// TIA Portal project "Pick_&_Place_XYZ_TIA_Portal" (V16)

(* hardware
DEVICE "S7-1200 station_1"  S7-1200 Station
   slot 0: "Rack_0"  S7-1200 Rack  Rack  V1.0
   slot 1: "PLC_1"  CPU 1215C DC/DC/DC  6ES7 215-1AG40-0XB0  V4.4
   slot 2: "DI 8x24VDC_1"  6ES7 221-1BF32-0XB0  V2.0
*)

// ===== PLC "PLC_1"  CPU 1215C DC/DC/DC =====

VAR_GLOBAL   // PLC tag table "Tabla de variables estándar"
   "pos_Y_alcanzada" AT %M0.6 : Bool;
   "pos_Z_alcanzada" AT %M0.7 : Bool;
   "Tag_1" AT %M500.3 : Bool;
   "Tag_2" AT %M200.0 : Bool;
   "arranque_cinta" AT %M1.0 : Bool;
END_VAR

VAR_GLOBAL   // PLC tag table "Entradas"
   "Box_at_place" AT %I2.0 : Bool;   // Sensor de posicion de lugar de carga del pale
   "Part_at_place" AT %I2.1 : Bool;   // Sensor de poscion de lugar de recogida de las cajas
   "Detected" AT %I2.2 : Bool;   // Sensor en la ventosa del robot cartesiano
   "C_limit" AT %I2.3 : Bool;   // Sensor que indica que la ventosa esta en angulo limite en giro en el eje Z
   "Start" AT %I2.4 : Bool;   // Pulsador de start
   "Reset" AT %I2.5 : Bool;   // Pulsador de reset
   "Stop" AT %I2.6 : Bool;   // Pulsador de stop
   "Emergency_stop" AT %I2.7 : Bool;   // Seta de emergencia
   "Auto" AT %I3.0 : Bool;   // Selector rotativo en posicion auto
   "X" AT %ID100 : Real;   // Coordenada X del robot, realimentada
   "Y" AT %ID104 : Real;   // Coordenada Y del robot, realimentada
   "Z" AT %ID108 : Real;   // Coordenada Z del robot, realimentada
END_VAR

VAR_GLOBAL   // PLC tag table "Salidas"
   "Box_conveyor" AT %Q0.0 : Bool;   // Cinta de rodillo para los pales
   "Part_conveyor" AT %Q0.1 : Bool;   // Cinta para las cajas
   "Exit_conveyor" AT %Q0.2 : Bool;   // Cinta de rodillo para salida de pales con cajas
   "C+" AT %Q0.3 : Bool;   // Actuador de giro de la ventosa, sentido horario mirando desde arriba
   "Grab" AT %Q0.4 : Bool;   // Ventosa
   "Exit_green" AT %Q0.5 : Bool;   // Semaforo industrial, color verde
   "Exit_yellow" AT %Q0.6 : Bool;   // Semaforo industrial, color amarillo
   "Exit_red" AT %Q0.7 : Bool;   // Semaforo industrial, color rojo
   "Start_light" AT %Q1.0 : Bool;   // Luz de pulsador de start
   "Reset_light" AT %Q1.1 : Bool;   // Luz de pulsador de reset
   "Stop_light" AT %Q1.2 : Bool;   // Luz de pulsador de stop
   "SP_X" AT %QD100 : Real;   // Salida de posicion del eje X del robot cartesiano
   "SP_Y" AT %QD104 : Real;   // Salida de posicion del eje Y del robot cartesiano
   "SP_Z" AT %QD108 : Real;   // Salida de posicion del eje Z del robor cartesiano
   "Counter" AT %QD112 : DInt;   // Display numerico para contador
END_VAR

VAR_GLOBAL   // PLC tag table "variables_auxiliares"
   "FlancoP_sensor_pales" AT %M10.0 : Bool;
   "Marcha" AT %M0.0 : Bool;
   "FlancoN_sensor_pales" AT %M500.0 : Bool;
   "Set_box_conveyor" AT %M500.1 : Bool;
   "FlancoP_estado_marcha" AT %M500.2 : Bool;
   "pale_terminado" AT %M0.1 : Bool;
   "Stop_filtrado" AT %M0.2 : Bool;
   "pos_X_alcanzada" AT %M0.5 : Bool;
   "caja_preparada" AT %M0.3 : Bool;
   "pale_preparado" AT %M0.4 : Bool;
END_VAR

TYPE "posicion_robot"
   STRUCT
      X : Real;
      Y : Real;
      Z : Real;
   END_STRUCT;
END_TYPE

// folder: DBs

DATA_BLOCK "contador_terminados_DB"   // DB1
{ S7_Optimized_Access := 'TRUE' }
VERSION : 0.1
// stored: InstanceOfName contador_terminados
"contador_terminados"
BEGIN
END_DATA_BLOCK

DATA_BLOCK "control_robot_y_ciclo_DB"   // DB2
{ S7_Optimized_Access := 'TRUE' }
VERSION : 0.1
// stored: InstanceOfName control_robot_y_ciclo
"control_robot_y_ciclo"
BEGIN
END_DATA_BLOCK

DATA_BLOCK "posiciones_robot"   // DB3
{ S7_Optimized_Access := 'TRUE' }
VERSION : 0.1
   VAR
      home : "posicion_robot";
      coger_caja_aprox : "posicion_robot";
      coger_caja : "posicion_robot";
      dejar_caja_1_aprox : "posicion_robot";
      dejar_caja_1 : "posicion_robot";
      dejar_caja_2_aprox : "posicion_robot";
      dejar_caja_2 : "posicion_robot";
      dejar_caja_3_aprox : "posicion_robot";
      dejar_caja_3 : "posicion_robot";
   END_VAR
BEGIN
   home.Y := 0.0;
   home.X := 0.0;
   home.Z := 0.0;
   coger_caja.X := 7.7;
   coger_caja.Y := 5.6;
   coger_caja.Z := 5.0;
   coger_caja_aprox.X := 7.7;
   coger_caja_aprox.Y := 5.6;
   coger_caja_aprox.Z := 0.0;
   dejar_caja_1_aprox.Y := 5.0;
   dejar_caja_1_aprox.Z := 0.0;
   dejar_caja_1.Z := 10.0;
   dejar_caja_1.Y := 5.0;
   dejar_caja_1_aprox.X := 2.5;
   dejar_caja_1.X := 2.5;
   dejar_caja_2.X := 4.2;
   dejar_caja_2.Y := 5.0;
   dejar_caja_2.Z := 10.0;
   dejar_caja_2_aprox.Z := 0.0;
   dejar_caja_2_aprox.Y := 5.0;
   dejar_caja_2_aprox.X := 4.2;
   dejar_caja_3.Y := 5.0;
   dejar_caja_3_aprox.Y := 5.0;
   dejar_caja_3_aprox.Z := 0.0;
   dejar_caja_3_aprox.X := 3.3;
   dejar_caja_3.X := 3.3;
   dejar_caja_3.Z := 5.5;
END_DATA_BLOCK

// folder: Conexion_factoryIO

FUNCTION "MHJ-PLC-Lab-Function-S71200" : Void   // FC9000, SCL
{ S7_Optimized_Access := 'TRUE' }
VERSION : 0.1
   VAR_TEMP
      rdTimeReturn : Int;
      outputTime : DTL;
      SyncVal : Byte;
      forVal : Int;
      forVal_2 : Int;
      Value : Byte;
   END_VAR
   VAR CONSTANT
      CompVal : Byte := 16#34;
      Value_01 : Byte := 16#11;
      Value_01_DW : DWord := 16#A165_D992;
      Value_02_DW : DWord := 16#58BE_4401;
   END_VAR
BEGIN

   #Value:=PEEK(area := 16#82,
        dbNumber := 0,
        byteOffset := 511);
   #Value := #Value + 1;

   POKE(area := 16#82,
        dbNumber := 0,
        byteOffset := 511,
        value := #Value);

   POKE(area:=16#81,
        dbNumber:=0,
        byteOffset:=1016,
        value:=#Value_01_DW);
   POKE(area := 16#81,
        dbNumber := 0,
        byteOffset := 1020,
        value := #Value_02_DW);

   POKE(area := 16#81,
        dbNumber := 0,
        byteOffset := 511,
        value := B#16#00);

   FOR #forVal := 0 TO 120 DO
       FOR #forVal_2:=0 TO 10 DO
           #rdTimeReturn:=RD_SYS_T(#outputTime);
           #rdTimeReturn := WR_SYS_T(#outputTime);
           #rdTimeReturn := RD_SYS_T(#outputTime);
           #rdTimeReturn := WR_SYS_T(#outputTime);
       END_FOR;
       #SyncVal:= PEEK(area := 16#81,
                      dbNumber := 0,
                      byteOffset := 511);
       IF #SyncVal = #CompVal THEN
          GOTO M_1;
       END_IF;
   END_FOR;
   RETURN;

   M_1:
   POKE(area := 16#81,
        dbNumber := 0,
        byteOffset := 511,
        value := B#16#0);
END_FUNCTION

// folder: FBs

FUNCTION_BLOCK "contador_terminados"   // FB1, LAD
{ S7_Optimized_Access := 'TRUE' }
VERSION : 0.1
   VAR RETAIN
      Contador_terminados : CTU_INT;
   END_VAR
   VAR_TEMP   // added for the SCL form of the ladder/FBD networks
      _w1 : Bool;
   END_VAR
BEGIN

REGION Network 1: Contador que incrementa con el flanco positivo de sesnsor NC, osea cuando el pale se va
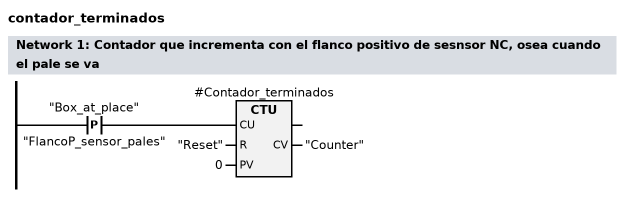
   #_w1 := "Box_at_place" AND NOT "FlancoP_sensor_pales";   // rising edge of "Box_at_place"
   "FlancoP_sensor_pales" := "Box_at_place";
   #Contador_terminados(CU := #_w1, R := "Reset", PV := 0, CV => "Counter");   // CTU
END_REGION
END_FUNCTION_BLOCK

FUNCTION_BLOCK "control_robot_y_ciclo"   // FB2, LAD
{ S7_Optimized_Access := 'TRUE' }
VERSION : 0.1
   VAR
      E0 : Bool;
      E1 : Bool;
      E2 : Bool;
      E3 : Bool;
      E4 : Bool;
      E5 : Bool;
      E6 : Bool;
      E7 : Bool;
      E8 : Bool;
      E9 : Bool;
      E10 : Bool;
      E11 : Bool;
      E12 : Bool;
      E13 : Bool;
      E14 : Bool;
      E15 : Bool;
      E16 : Bool;
      E17 : Bool;
      E18 : Bool;
      E19 : Bool;
      E20 : Bool;
      E21 : Bool;
      E22 : Bool;
      pos_X_alcanzada : Bool;
      pos_Y_alcanzada : Bool;
      pos_Z_alcanzada : Bool;
      aux1 : Bool;
      aux2 : Bool;
      aux3 : Bool;
      aux4 : Bool;
      aux5 : Bool;
      TON_1 : TON_TIME;
      TON_2 : TON_TIME;
      TON_3 : TON_TIME;
      TON_4 : TON_TIME;
   END_VAR
   VAR_TEMP   // added for the SCL form of the ladder/FBD networks
      _w1 : Bool;
      _w2 : Bool;
      _w3 : Bool;
      _w4 : Bool;
      _w5 : Bool;
      _w6 : Bool;
      _w7 : Bool;
   END_VAR
BEGIN

REGION Network 1
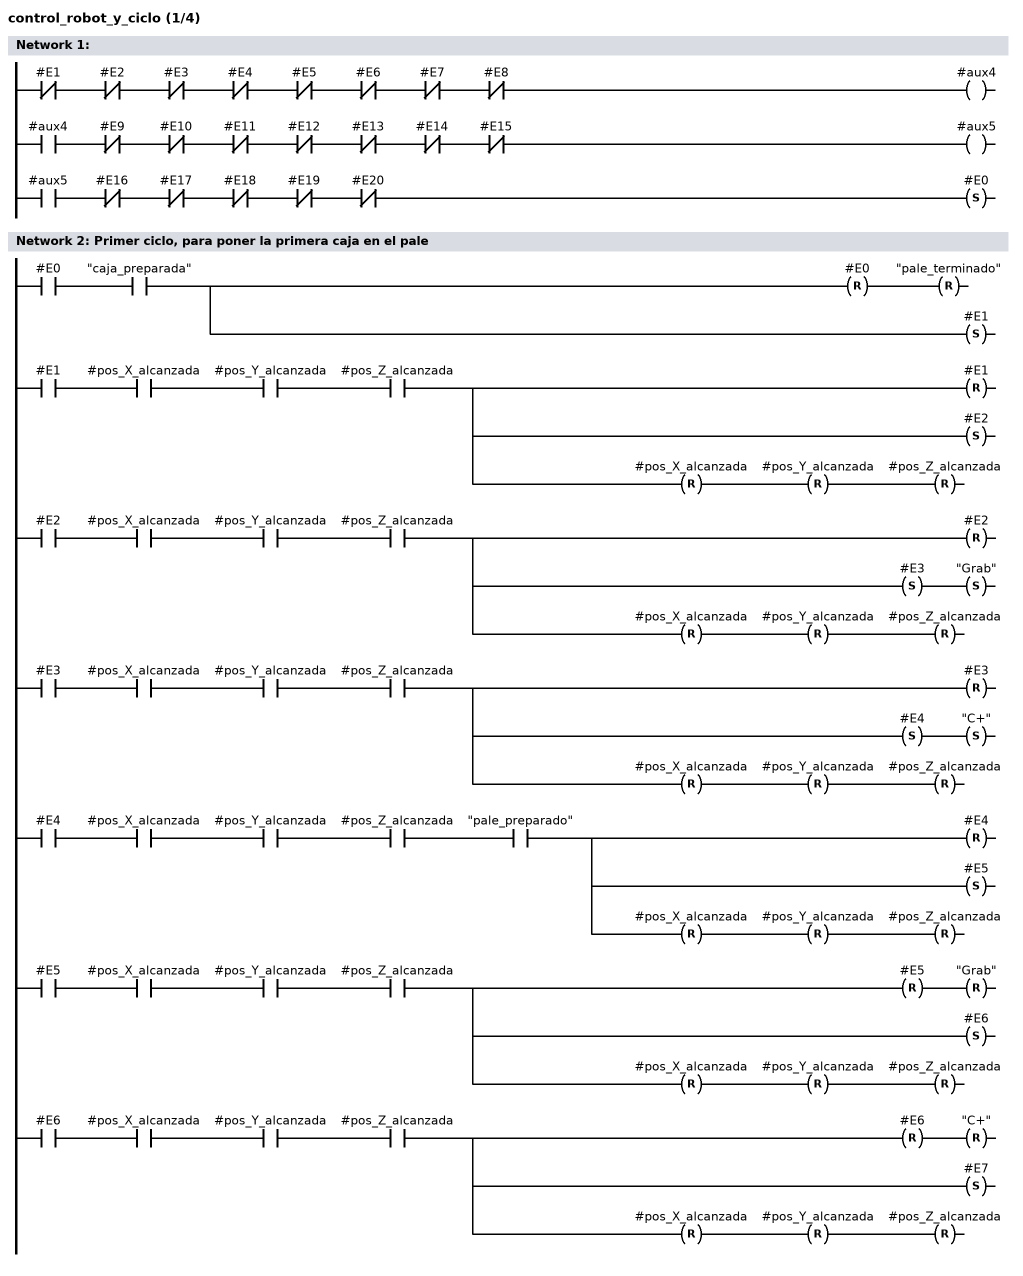
   RUNG wire#powerrail
      I_Contact( #E1 )
      I_Contact( #E2 )
      I_Contact( #E3 )
      I_Contact( #E4 )
      I_Contact( #E5 )
      I_Contact( #E6 )
      I_Contact( #E7 )
      I_Contact( #E8 )
      Coil( #aux4 )
   END_RUNG
   RUNG wire#powerrail
      Contact( #aux4 )
      I_Contact( #E9 )
      I_Contact( #E10 )
      I_Contact( #E11 )
      I_Contact( #E12 )
      I_Contact( #E13 )
      I_Contact( #E14 )
      I_Contact( #E15 )
      Coil( #aux5 )
   END_RUNG
   RUNG wire#powerrail
      Contact( #aux5 )
      I_Contact( #E16 )
      I_Contact( #E17 )
      I_Contact( #E18 )
      I_Contact( #E19 )
      I_Contact( #E20 )
      S_Coil( #E0 )
   END_RUNG
   // the same network as SCL:
   #aux4 := NOT #E1 AND NOT #E2 AND NOT #E3 AND NOT #E4 AND NOT #E5 AND NOT #E6 AND NOT #E7 AND NOT #E8;
   #aux5 := #aux4 AND NOT #E9 AND NOT #E10 AND NOT #E11 AND NOT #E12 AND NOT #E13 AND NOT #E14 AND NOT #E15;
   IF #aux5 AND NOT #E16 AND NOT #E17 AND NOT #E18 AND NOT #E19 AND NOT #E20 THEN #E0 := TRUE; END_IF;
END_REGION

REGION Network 2: Primer ciclo, para poner la primera caja en el pale
   RUNG wire#powerrail
      Contact( #E0 )
      Contact( "caja_preparada" )
      wire#w1
      R_Coil( #E0 )
      R_Coil( "pale_terminado" )
   END_RUNG
   RUNG wire#w1
      S_Coil( #E1 )
   END_RUNG
   RUNG wire#powerrail
      Contact( #E1 )
      Contact( #pos_X_alcanzada )
      Contact( #pos_Y_alcanzada )
      Contact( #pos_Z_alcanzada )
      wire#w2
      R_Coil( #E1 )
   END_RUNG
   RUNG wire#w2
      S_Coil( #E2 )
   END_RUNG
   RUNG wire#w2
      R_Coil( #pos_X_alcanzada )
      R_Coil( #pos_Y_alcanzada )
      R_Coil( #pos_Z_alcanzada )
   END_RUNG
   RUNG wire#powerrail
      Contact( #E2 )
      Contact( #pos_X_alcanzada )
      Contact( #pos_Y_alcanzada )
      Contact( #pos_Z_alcanzada )
      wire#w3
      R_Coil( #E2 )
   END_RUNG
   RUNG wire#w3
      S_Coil( #E3 )
      S_Coil( "Grab" )
   END_RUNG
   RUNG wire#w3
      R_Coil( #pos_X_alcanzada )
      R_Coil( #pos_Y_alcanzada )
      R_Coil( #pos_Z_alcanzada )
   END_RUNG
   RUNG wire#powerrail
      Contact( #E3 )
      Contact( #pos_X_alcanzada )
      Contact( #pos_Y_alcanzada )
      Contact( #pos_Z_alcanzada )
      wire#w4
      R_Coil( #E3 )
   END_RUNG
   RUNG wire#w4
      S_Coil( #E4 )
      S_Coil( "C+" )
   END_RUNG
   RUNG wire#w4
      R_Coil( #pos_X_alcanzada )
      R_Coil( #pos_Y_alcanzada )
      R_Coil( #pos_Z_alcanzada )
   END_RUNG
   RUNG wire#powerrail
      Contact( #E4 )
      Contact( #pos_X_alcanzada )
      Contact( #pos_Y_alcanzada )
      Contact( #pos_Z_alcanzada )
      Contact( "pale_preparado" )
      wire#w5
      R_Coil( #E4 )
   END_RUNG
   RUNG wire#w5
      S_Coil( #E5 )
   END_RUNG
   RUNG wire#w5
      R_Coil( #pos_X_alcanzada )
      R_Coil( #pos_Y_alcanzada )
      R_Coil( #pos_Z_alcanzada )
   END_RUNG
   RUNG wire#powerrail
      Contact( #E5 )
      Contact( #pos_X_alcanzada )
      Contact( #pos_Y_alcanzada )
      Contact( #pos_Z_alcanzada )
      wire#w6
      R_Coil( #E5 )
      R_Coil( "Grab" )
   END_RUNG
   RUNG wire#w6
      S_Coil( #E6 )
   END_RUNG
   RUNG wire#w6
      R_Coil( #pos_X_alcanzada )
      R_Coil( #pos_Y_alcanzada )
      R_Coil( #pos_Z_alcanzada )
   END_RUNG
   RUNG wire#powerrail
      Contact( #E6 )
      Contact( #pos_X_alcanzada )
      Contact( #pos_Y_alcanzada )
      Contact( #pos_Z_alcanzada )
      wire#w7
      R_Coil( #E6 )
      R_Coil( "C+" )
   END_RUNG
   RUNG wire#w7
      S_Coil( #E7 )
   END_RUNG
   RUNG wire#w7
      R_Coil( #pos_X_alcanzada )
      R_Coil( #pos_Y_alcanzada )
      R_Coil( #pos_Z_alcanzada )
   END_RUNG
   // the same network as SCL:
   #_w1 := #E0 AND "caja_preparada";
   IF #_w1 THEN
       #E0 := FALSE;
       "pale_terminado" := FALSE;
       #E1 := TRUE;
   END_IF;
   #_w2 := #E1 AND #pos_X_alcanzada AND #pos_Y_alcanzada AND #pos_Z_alcanzada;
   IF #_w2 THEN
       #E1 := FALSE;
       #E2 := TRUE;
       #pos_X_alcanzada := FALSE;
       #pos_Y_alcanzada := FALSE;
       #pos_Z_alcanzada := FALSE;
   END_IF;
   #_w3 := #E2 AND #pos_X_alcanzada AND #pos_Y_alcanzada AND #pos_Z_alcanzada;
   IF #_w3 THEN
       #E2 := FALSE;
       #E3 := TRUE;
       "Grab" := TRUE;
       #pos_X_alcanzada := FALSE;
       #pos_Y_alcanzada := FALSE;
       #pos_Z_alcanzada := FALSE;
   END_IF;
   #_w4 := #E3 AND #pos_X_alcanzada AND #pos_Y_alcanzada AND #pos_Z_alcanzada;
   IF #_w4 THEN
       #E3 := FALSE;
       #E4 := TRUE;
       "C+" := TRUE;
       #pos_X_alcanzada := FALSE;
       #pos_Y_alcanzada := FALSE;
       #pos_Z_alcanzada := FALSE;
   END_IF;
   #_w5 := #E4 AND #pos_X_alcanzada AND #pos_Y_alcanzada AND #pos_Z_alcanzada AND "pale_preparado";
   IF #_w5 THEN
       #E4 := FALSE;
       #E5 := TRUE;
       #pos_X_alcanzada := FALSE;
       #pos_Y_alcanzada := FALSE;
       #pos_Z_alcanzada := FALSE;
   END_IF;
   #_w6 := #E5 AND #pos_X_alcanzada AND #pos_Y_alcanzada AND #pos_Z_alcanzada;
   IF #_w6 THEN
       #E5 := FALSE;
       "Grab" := FALSE;
       #E6 := TRUE;
       #pos_X_alcanzada := FALSE;
       #pos_Y_alcanzada := FALSE;
       #pos_Z_alcanzada := FALSE;
   END_IF;
   #_w7 := #E6 AND #pos_X_alcanzada AND #pos_Y_alcanzada AND #pos_Z_alcanzada;
   IF #_w7 THEN
       #E6 := FALSE;
       "C+" := FALSE;
       #E7 := TRUE;
       #pos_X_alcanzada := FALSE;
       #pos_Y_alcanzada := FALSE;
       #pos_Z_alcanzada := FALSE;
   END_IF;
END_REGION

REGION Network 3: segundo ciclo, para poner la segunda caja en el pale
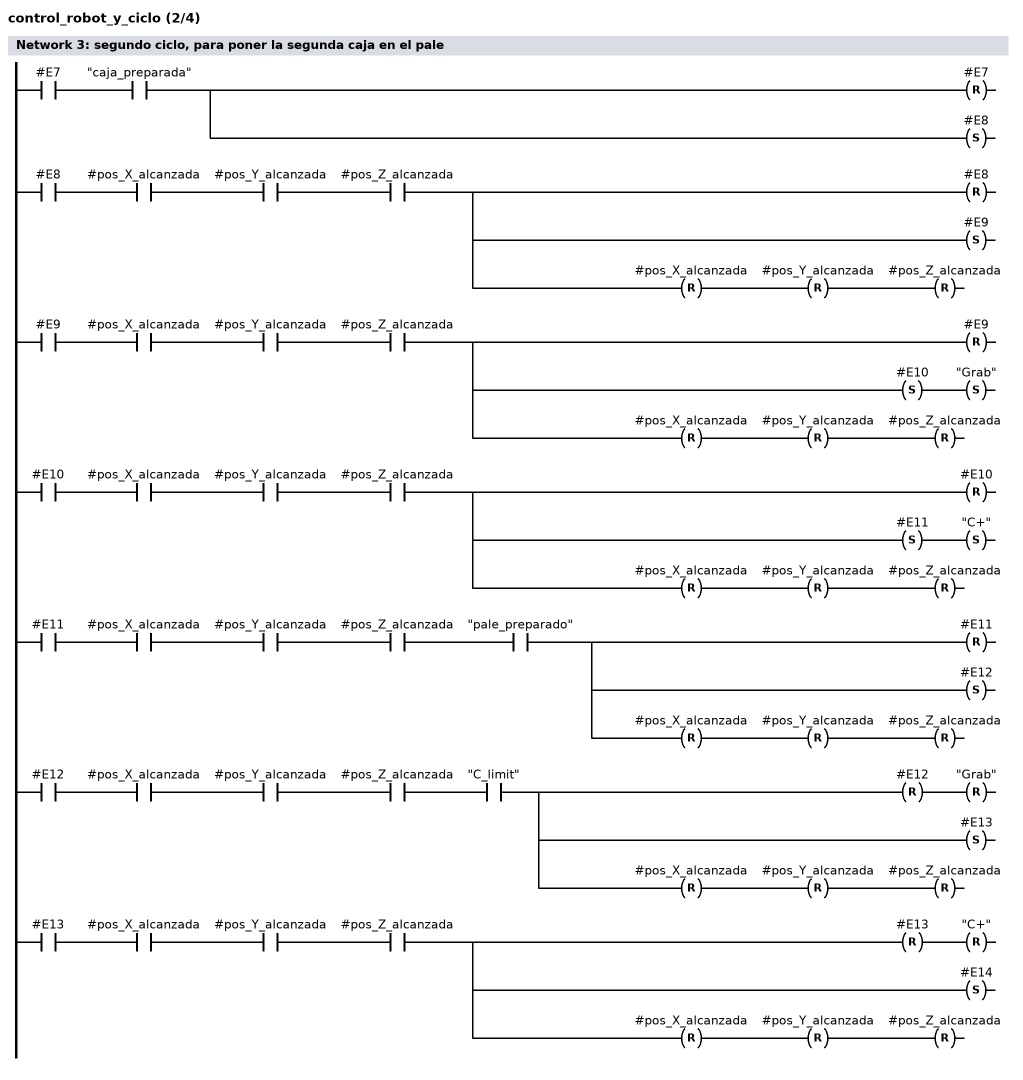
   RUNG wire#powerrail
      Contact( #E7 )
      Contact( "caja_preparada" )
      wire#w1
      R_Coil( #E7 )
   END_RUNG
   RUNG wire#w1
      S_Coil( #E8 )
   END_RUNG
   RUNG wire#powerrail
      Contact( #E8 )
      Contact( #pos_X_alcanzada )
      Contact( #pos_Y_alcanzada )
      Contact( #pos_Z_alcanzada )
      wire#w2
      R_Coil( #E8 )
   END_RUNG
   RUNG wire#w2
      S_Coil( #E9 )
   END_RUNG
   RUNG wire#w2
      R_Coil( #pos_X_alcanzada )
      R_Coil( #pos_Y_alcanzada )
      R_Coil( #pos_Z_alcanzada )
   END_RUNG
   RUNG wire#powerrail
      Contact( #E9 )
      Contact( #pos_X_alcanzada )
      Contact( #pos_Y_alcanzada )
      Contact( #pos_Z_alcanzada )
      wire#w3
      R_Coil( #E9 )
   END_RUNG
   RUNG wire#w3
      S_Coil( #E10 )
      S_Coil( "Grab" )
   END_RUNG
   RUNG wire#w3
      R_Coil( #pos_X_alcanzada )
      R_Coil( #pos_Y_alcanzada )
      R_Coil( #pos_Z_alcanzada )
   END_RUNG
   RUNG wire#powerrail
      Contact( #E10 )
      Contact( #pos_X_alcanzada )
      Contact( #pos_Y_alcanzada )
      Contact( #pos_Z_alcanzada )
      wire#w4
      R_Coil( #E10 )
   END_RUNG
   RUNG wire#w4
      S_Coil( #E11 )
      S_Coil( "C+" )
   END_RUNG
   RUNG wire#w4
      R_Coil( #pos_X_alcanzada )
      R_Coil( #pos_Y_alcanzada )
      R_Coil( #pos_Z_alcanzada )
   END_RUNG
   RUNG wire#powerrail
      Contact( #E11 )
      Contact( #pos_X_alcanzada )
      Contact( #pos_Y_alcanzada )
      Contact( #pos_Z_alcanzada )
      Contact( "pale_preparado" )
      wire#w5
      R_Coil( #E11 )
   END_RUNG
   RUNG wire#w5
      S_Coil( #E12 )
   END_RUNG
   RUNG wire#w5
      R_Coil( #pos_X_alcanzada )
      R_Coil( #pos_Y_alcanzada )
      R_Coil( #pos_Z_alcanzada )
   END_RUNG
   RUNG wire#powerrail
      Contact( #E12 )
      Contact( #pos_X_alcanzada )
      Contact( #pos_Y_alcanzada )
      Contact( #pos_Z_alcanzada )
      Contact( "C_limit" )
      wire#w6
      R_Coil( #E12 )
      R_Coil( "Grab" )
   END_RUNG
   RUNG wire#w6
      S_Coil( #E13 )
   END_RUNG
   RUNG wire#w6
      R_Coil( #pos_X_alcanzada )
      R_Coil( #pos_Y_alcanzada )
      R_Coil( #pos_Z_alcanzada )
   END_RUNG
   RUNG wire#powerrail
      Contact( #E13 )
      Contact( #pos_X_alcanzada )
      Contact( #pos_Y_alcanzada )
      Contact( #pos_Z_alcanzada )
      wire#w7
      R_Coil( #E13 )
      R_Coil( "C+" )
   END_RUNG
   RUNG wire#w7
      S_Coil( #E14 )
   END_RUNG
   RUNG wire#w7
      R_Coil( #pos_X_alcanzada )
      R_Coil( #pos_Y_alcanzada )
      R_Coil( #pos_Z_alcanzada )
   END_RUNG
   // the same network as SCL:
   #_w1 := #E7 AND "caja_preparada";
   IF #_w1 THEN
       #E7 := FALSE;
       #E8 := TRUE;
   END_IF;
   #_w2 := #E8 AND #pos_X_alcanzada AND #pos_Y_alcanzada AND #pos_Z_alcanzada;
   IF #_w2 THEN
       #E8 := FALSE;
       #E9 := TRUE;
       #pos_X_alcanzada := FALSE;
       #pos_Y_alcanzada := FALSE;
       #pos_Z_alcanzada := FALSE;
   END_IF;
   #_w3 := #E9 AND #pos_X_alcanzada AND #pos_Y_alcanzada AND #pos_Z_alcanzada;
   IF #_w3 THEN
       #E9 := FALSE;
       #E10 := TRUE;
       "Grab" := TRUE;
       #pos_X_alcanzada := FALSE;
       #pos_Y_alcanzada := FALSE;
       #pos_Z_alcanzada := FALSE;
   END_IF;
   #_w4 := #E10 AND #pos_X_alcanzada AND #pos_Y_alcanzada AND #pos_Z_alcanzada;
   IF #_w4 THEN
       #E10 := FALSE;
       #E11 := TRUE;
       "C+" := TRUE;
       #pos_X_alcanzada := FALSE;
       #pos_Y_alcanzada := FALSE;
       #pos_Z_alcanzada := FALSE;
   END_IF;
   #_w5 := #E11 AND #pos_X_alcanzada AND #pos_Y_alcanzada AND #pos_Z_alcanzada AND "pale_preparado";
   IF #_w5 THEN
       #E11 := FALSE;
       #E12 := TRUE;
       #pos_X_alcanzada := FALSE;
       #pos_Y_alcanzada := FALSE;
       #pos_Z_alcanzada := FALSE;
   END_IF;
   #_w6 := #E12 AND #pos_X_alcanzada AND #pos_Y_alcanzada AND #pos_Z_alcanzada AND "C_limit";
   IF #_w6 THEN
       #E12 := FALSE;
       "Grab" := FALSE;
       #E13 := TRUE;
       #pos_X_alcanzada := FALSE;
       #pos_Y_alcanzada := FALSE;
       #pos_Z_alcanzada := FALSE;
   END_IF;
   #_w7 := #E13 AND #pos_X_alcanzada AND #pos_Y_alcanzada AND #pos_Z_alcanzada;
   IF #_w7 THEN
       #E13 := FALSE;
       "C+" := FALSE;
       #E14 := TRUE;
       #pos_X_alcanzada := FALSE;
       #pos_Y_alcanzada := FALSE;
       #pos_Z_alcanzada := FALSE;
   END_IF;
END_REGION

REGION Network 4: segundo ciclo, para poner la segunda caja en el pale
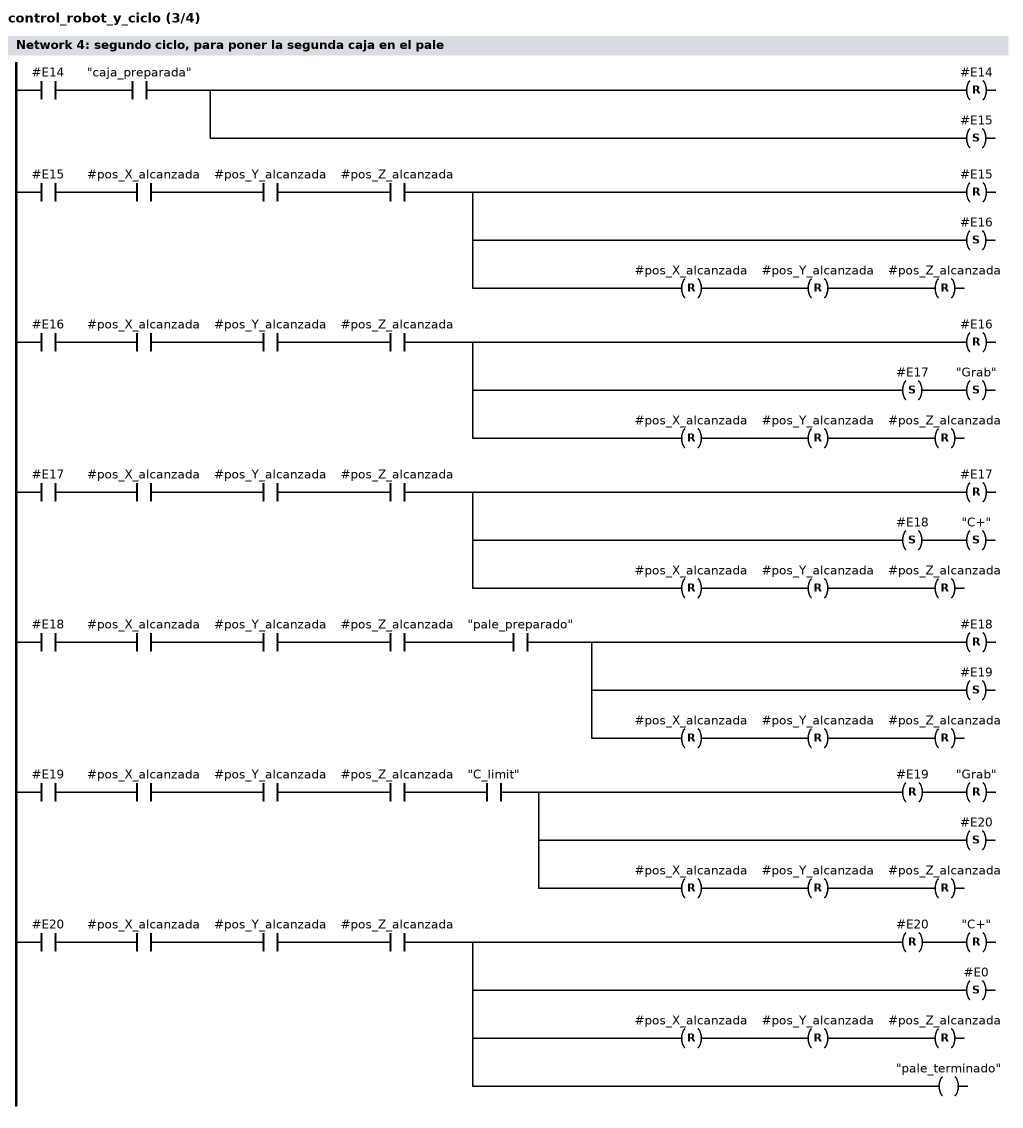
   RUNG wire#powerrail
      Contact( #E14 )
      Contact( "caja_preparada" )
      wire#w1
      R_Coil( #E14 )
   END_RUNG
   RUNG wire#w1
      S_Coil( #E15 )
   END_RUNG
   RUNG wire#powerrail
      Contact( #E15 )
      Contact( #pos_X_alcanzada )
      Contact( #pos_Y_alcanzada )
      Contact( #pos_Z_alcanzada )
      wire#w2
      R_Coil( #E15 )
   END_RUNG
   RUNG wire#w2
      S_Coil( #E16 )
   END_RUNG
   RUNG wire#w2
      R_Coil( #pos_X_alcanzada )
      R_Coil( #pos_Y_alcanzada )
      R_Coil( #pos_Z_alcanzada )
   END_RUNG
   RUNG wire#powerrail
      Contact( #E16 )
      Contact( #pos_X_alcanzada )
      Contact( #pos_Y_alcanzada )
      Contact( #pos_Z_alcanzada )
      wire#w3
      R_Coil( #E16 )
   END_RUNG
   RUNG wire#w3
      S_Coil( #E17 )
      S_Coil( "Grab" )
   END_RUNG
   RUNG wire#w3
      R_Coil( #pos_X_alcanzada )
      R_Coil( #pos_Y_alcanzada )
      R_Coil( #pos_Z_alcanzada )
   END_RUNG
   RUNG wire#powerrail
      Contact( #E17 )
      Contact( #pos_X_alcanzada )
      Contact( #pos_Y_alcanzada )
      Contact( #pos_Z_alcanzada )
      wire#w4
      R_Coil( #E17 )
   END_RUNG
   RUNG wire#w4
      S_Coil( #E18 )
      S_Coil( "C+" )
   END_RUNG
   RUNG wire#w4
      R_Coil( #pos_X_alcanzada )
      R_Coil( #pos_Y_alcanzada )
      R_Coil( #pos_Z_alcanzada )
   END_RUNG
   RUNG wire#powerrail
      Contact( #E18 )
      Contact( #pos_X_alcanzada )
      Contact( #pos_Y_alcanzada )
      Contact( #pos_Z_alcanzada )
      Contact( "pale_preparado" )
      wire#w5
      R_Coil( #E18 )
   END_RUNG
   RUNG wire#w5
      S_Coil( #E19 )
   END_RUNG
   RUNG wire#w5
      R_Coil( #pos_X_alcanzada )
      R_Coil( #pos_Y_alcanzada )
      R_Coil( #pos_Z_alcanzada )
   END_RUNG
   RUNG wire#powerrail
      Contact( #E19 )
      Contact( #pos_X_alcanzada )
      Contact( #pos_Y_alcanzada )
      Contact( #pos_Z_alcanzada )
      Contact( "C_limit" )
      wire#w6
      R_Coil( #E19 )
      R_Coil( "Grab" )
   END_RUNG
   RUNG wire#w6
      S_Coil( #E20 )
   END_RUNG
   RUNG wire#w6
      R_Coil( #pos_X_alcanzada )
      R_Coil( #pos_Y_alcanzada )
      R_Coil( #pos_Z_alcanzada )
   END_RUNG
   RUNG wire#powerrail
      Contact( #E20 )
      Contact( #pos_X_alcanzada )
      Contact( #pos_Y_alcanzada )
      Contact( #pos_Z_alcanzada )
      wire#w7
      R_Coil( #E20 )
      R_Coil( "C+" )
   END_RUNG
   RUNG wire#w7
      S_Coil( #E0 )
   END_RUNG
   RUNG wire#w7
      R_Coil( #pos_X_alcanzada )
      R_Coil( #pos_Y_alcanzada )
      R_Coil( #pos_Z_alcanzada )
   END_RUNG
   RUNG wire#w7
      Coil( "pale_terminado" )
   END_RUNG
   // the same network as SCL:
   #_w1 := #E14 AND "caja_preparada";
   IF #_w1 THEN
       #E14 := FALSE;
       #E15 := TRUE;
   END_IF;
   #_w2 := #E15 AND #pos_X_alcanzada AND #pos_Y_alcanzada AND #pos_Z_alcanzada;
   IF #_w2 THEN
       #E15 := FALSE;
       #E16 := TRUE;
       #pos_X_alcanzada := FALSE;
       #pos_Y_alcanzada := FALSE;
       #pos_Z_alcanzada := FALSE;
   END_IF;
   #_w3 := #E16 AND #pos_X_alcanzada AND #pos_Y_alcanzada AND #pos_Z_alcanzada;
   IF #_w3 THEN
       #E16 := FALSE;
       #E17 := TRUE;
       "Grab" := TRUE;
       #pos_X_alcanzada := FALSE;
       #pos_Y_alcanzada := FALSE;
       #pos_Z_alcanzada := FALSE;
   END_IF;
   #_w4 := #E17 AND #pos_X_alcanzada AND #pos_Y_alcanzada AND #pos_Z_alcanzada;
   IF #_w4 THEN
       #E17 := FALSE;
       #E18 := TRUE;
       "C+" := TRUE;
       #pos_X_alcanzada := FALSE;
       #pos_Y_alcanzada := FALSE;
       #pos_Z_alcanzada := FALSE;
   END_IF;
   #_w5 := #E18 AND #pos_X_alcanzada AND #pos_Y_alcanzada AND #pos_Z_alcanzada AND "pale_preparado";
   IF #_w5 THEN
       #E18 := FALSE;
       #E19 := TRUE;
       #pos_X_alcanzada := FALSE;
       #pos_Y_alcanzada := FALSE;
       #pos_Z_alcanzada := FALSE;
   END_IF;
   #_w6 := #E19 AND #pos_X_alcanzada AND #pos_Y_alcanzada AND #pos_Z_alcanzada AND "C_limit";
   IF #_w6 THEN
       #E19 := FALSE;
       "Grab" := FALSE;
       #E20 := TRUE;
       #pos_X_alcanzada := FALSE;
       #pos_Y_alcanzada := FALSE;
       #pos_Z_alcanzada := FALSE;
   END_IF;
   #_w7 := #E20 AND #pos_X_alcanzada AND #pos_Y_alcanzada AND #pos_Z_alcanzada;
   IF #_w7 THEN
       #E20 := FALSE;
       "C+" := FALSE;
       #E0 := TRUE;
       #pos_X_alcanzada := FALSE;
       #pos_Y_alcanzada := FALSE;
       #pos_Z_alcanzada := FALSE;
   END_IF;
   "pale_terminado" := #_w7;
END_REGION

REGION Network 5: Actuador de giro de la ventosa, sentido horario mirando desde arriba
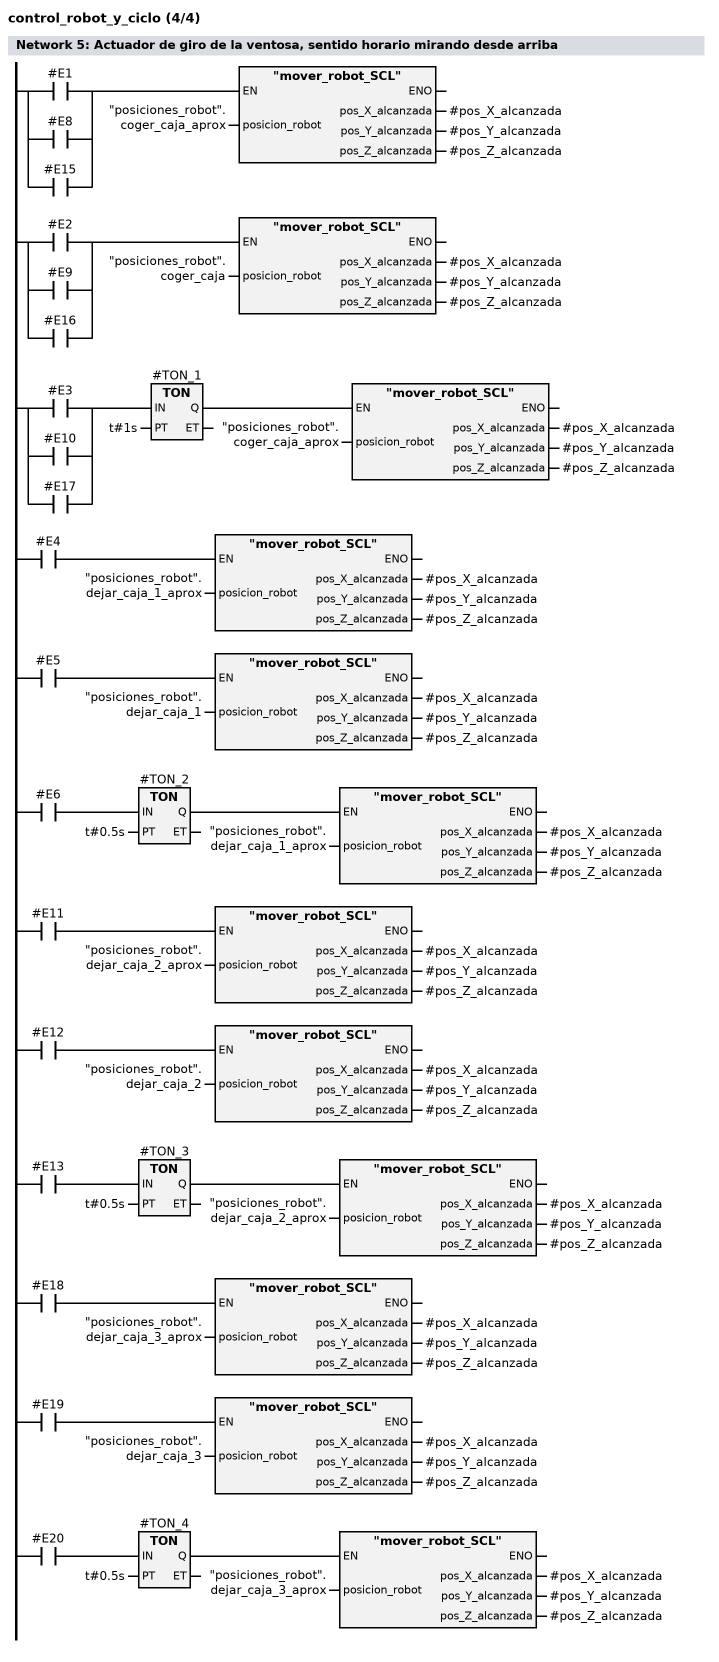
   IF #E1 OR #E8 OR #E15 THEN
       "mover_robot_SCL"(posicion_robot := "posiciones_robot".coger_caja_aprox,
                         pos_X_alcanzada => #pos_X_alcanzada,
                         pos_Y_alcanzada => #pos_Y_alcanzada,
                         pos_Z_alcanzada => #pos_Z_alcanzada);
   END_IF;
   IF #E2 OR #E9 OR #E16 THEN
       "mover_robot_SCL"(posicion_robot := "posiciones_robot".coger_caja,
                         pos_X_alcanzada => #pos_X_alcanzada,
                         pos_Y_alcanzada => #pos_Y_alcanzada,
                         pos_Z_alcanzada => #pos_Z_alcanzada);
   END_IF;
   #TON_1(IN := #E3 OR #E10 OR #E17, PT := t#1s);   // TON
   IF #TON_1.Q THEN
       "mover_robot_SCL"(posicion_robot := "posiciones_robot".coger_caja_aprox,
                         pos_X_alcanzada => #pos_X_alcanzada,
                         pos_Y_alcanzada => #pos_Y_alcanzada,
                         pos_Z_alcanzada => #pos_Z_alcanzada);
   END_IF;
   IF #E4 THEN
       "mover_robot_SCL"(posicion_robot := "posiciones_robot".dejar_caja_1_aprox,
                         pos_X_alcanzada => #pos_X_alcanzada,
                         pos_Y_alcanzada => #pos_Y_alcanzada,
                         pos_Z_alcanzada => #pos_Z_alcanzada);
   END_IF;
   IF #E5 THEN
       "mover_robot_SCL"(posicion_robot := "posiciones_robot".dejar_caja_1,
                         pos_X_alcanzada => #pos_X_alcanzada,
                         pos_Y_alcanzada => #pos_Y_alcanzada,
                         pos_Z_alcanzada => #pos_Z_alcanzada);
   END_IF;
   #TON_2(IN := #E6, PT := t#0.5s);   // TON
   IF #TON_2.Q THEN
       "mover_robot_SCL"(posicion_robot := "posiciones_robot".dejar_caja_1_aprox,
                         pos_X_alcanzada => #pos_X_alcanzada,
                         pos_Y_alcanzada => #pos_Y_alcanzada,
                         pos_Z_alcanzada => #pos_Z_alcanzada);
   END_IF;
   IF #E11 THEN
       "mover_robot_SCL"(posicion_robot := "posiciones_robot".dejar_caja_2_aprox,
                         pos_X_alcanzada => #pos_X_alcanzada,
                         pos_Y_alcanzada => #pos_Y_alcanzada,
                         pos_Z_alcanzada => #pos_Z_alcanzada);
   END_IF;
   IF #E12 THEN
       "mover_robot_SCL"(posicion_robot := "posiciones_robot".dejar_caja_2,
                         pos_X_alcanzada => #pos_X_alcanzada,
                         pos_Y_alcanzada => #pos_Y_alcanzada,
                         pos_Z_alcanzada => #pos_Z_alcanzada);
   END_IF;
   #TON_3(IN := #E13, PT := t#0.5s);   // TON
   IF #TON_3.Q THEN
       "mover_robot_SCL"(posicion_robot := "posiciones_robot".dejar_caja_2_aprox,
                         pos_X_alcanzada => #pos_X_alcanzada,
                         pos_Y_alcanzada => #pos_Y_alcanzada,
                         pos_Z_alcanzada => #pos_Z_alcanzada);
   END_IF;
   IF #E18 THEN
       "mover_robot_SCL"(posicion_robot := "posiciones_robot".dejar_caja_3_aprox,
                         pos_X_alcanzada => #pos_X_alcanzada,
                         pos_Y_alcanzada => #pos_Y_alcanzada,
                         pos_Z_alcanzada => #pos_Z_alcanzada);
   END_IF;
   IF #E19 THEN
       "mover_robot_SCL"(posicion_robot := "posiciones_robot".dejar_caja_3,
                         pos_X_alcanzada => #pos_X_alcanzada,
                         pos_Y_alcanzada => #pos_Y_alcanzada,
                         pos_Z_alcanzada => #pos_Z_alcanzada);
   END_IF;
   #TON_4(IN := #E20, PT := t#0.5s);   // TON
   IF #TON_4.Q THEN
       "mover_robot_SCL"(posicion_robot := "posiciones_robot".dejar_caja_3_aprox,
                         pos_X_alcanzada => #pos_X_alcanzada,
                         pos_Y_alcanzada => #pos_Y_alcanzada,
                         pos_Z_alcanzada => #pos_Z_alcanzada);
   END_IF;
END_REGION
END_FUNCTION_BLOCK

// folder: FCs

FUNCTION "luces_botones" : Void   // FC1, LAD
{ S7_Optimized_Access := 'TRUE' }
VERSION : 0.1
BEGIN

REGION Network 1: Luz de pulsador de start
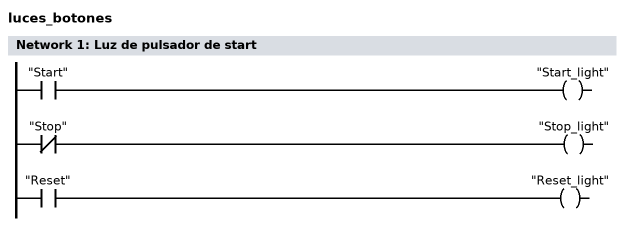
   RUNG wire#powerrail
      Contact( "Start" )
      Coil( "Start_light" )
   END_RUNG
   RUNG wire#powerrail
      I_Contact( "Stop" )
      Coil( "Stop_light" )
   END_RUNG
   RUNG wire#powerrail
      Contact( "Reset" )
      Coil( "Reset_light" )
   END_RUNG
   // the same network as SCL:
   "Start_light" := "Start";
   "Stop_light" := NOT "Stop";
   "Reset_light" := "Reset";
END_REGION
END_FUNCTION

FUNCTION "Control_cinta_cajas" : Void   // FC2, LAD
{ S7_Optimized_Access := 'TRUE' }
VERSION : 0.1
   VAR_OUTPUT
      caja_en_posicion : Bool;
   END_VAR
BEGIN

REGION Network 1: Cinta de rodillo para los pales
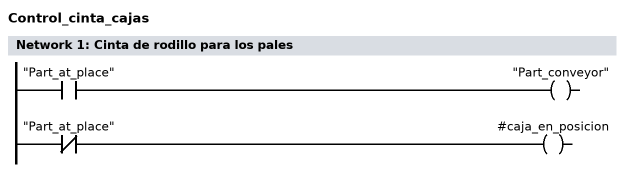
   RUNG wire#powerrail
      Contact( "Part_at_place" )
      Coil( "Part_conveyor" )
   END_RUNG
   RUNG wire#powerrail
      I_Contact( "Part_at_place" )
      Coil( #caja_en_posicion )
   END_RUNG
   // the same network as SCL:
   "Part_conveyor" := "Part_at_place";
   #caja_en_posicion := NOT "Part_at_place";
END_REGION
END_FUNCTION

FUNCTION "Control_exit_conveyor" : Void   // FC4, LAD
{ S7_Optimized_Access := 'TRUE' }
VERSION : 0.1
BEGIN

REGION Network 1: Cinta de rodillo para salida de pales con cajas
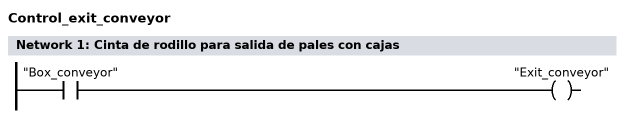
   RUNG wire#powerrail
      Contact( "Box_conveyor" )
      Coil( "Exit_conveyor" )
   END_RUNG
   // the same network as SCL:
   "Exit_conveyor" := "Box_conveyor";
END_REGION
END_FUNCTION

FUNCTION "Control_cinta_entrada" : Void   // FC5, LAD
{ S7_Optimized_Access := 'TRUE' }
VERSION : 0.1
   VAR_OUTPUT
      pale_en_posicion : Bool;
   END_VAR
   VAR_TEMP   // added for the SCL form of the ladder/FBD networks
      _w1 : Bool;
   END_VAR
BEGIN

REGION Network 1: Cinta de rodillo para los pales
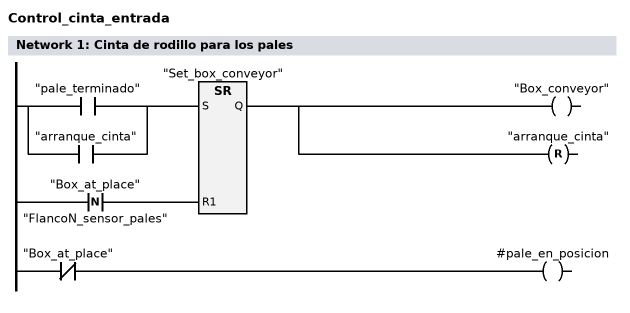
   RUNG wire#powerrail
      Contact( "pale_terminado" )
      wire#w1
      S_SR(operand := "Set_box_conveyor", r1 := wire#w2)
      wire#w3
      Coil( "Box_conveyor" )
   END_RUNG
   RUNG wire#powerrail
      Contact( "arranque_cinta" )
   END_RUNG wire#w1
   RUNG wire#powerrail
      N_Contact(operand := "Box_at_place", bit := "FlancoN_sensor_pales")
   END_RUNG wire#w2
   RUNG wire#w3
      R_Coil( "arranque_cinta" )
   END_RUNG
   RUNG wire#powerrail
      I_Contact( "Box_at_place" )
      Coil( #pale_en_posicion )
   END_RUNG
   // the same network as SCL:
   #_w1 := NOT "Box_at_place" AND "FlancoN_sensor_pales";   // falling edge of "Box_at_place"
   "FlancoN_sensor_pales" := "Box_at_place";
   IF "pale_terminado" OR "arranque_cinta" THEN
       "Set_box_conveyor" := TRUE;   // SR flip-flop
   END_IF;
   IF #_w1 THEN "Set_box_conveyor" := FALSE; END_IF;
   "Box_conveyor" := "Set_box_conveyor";
   IF "Set_box_conveyor" THEN "arranque_cinta" := FALSE; END_IF;
   #pale_en_posicion := NOT "Box_at_place";
END_REGION
END_FUNCTION

FUNCTION "mover_robot_SCL" : Void   // FC6, SCL
{ S7_Optimized_Access := 'TRUE' }
VERSION : 0.1
   VAR_INPUT
      posicion_robot : "posicion_robot";
   END_VAR
   VAR_OUTPUT
      pos_X_alcanzada : Bool;
      pos_Y_alcanzada : Bool;
      pos_Z_alcanzada : Bool;
   END_VAR
BEGIN
   "SP_X" := #posicion_robot.X;
   "SP_Y" := #posicion_robot.Y;
   "SP_Z" := #posicion_robot.Z;

   IF ("X">= ("SP_X" - 0.01)) AND ("X" <= ("SP_X" + 0.01)) THEN
       #pos_X_alcanzada := true;
   END_IF;

   IF ("Y">= ("SP_Y"- 0.01)) AND ("Y"<= ("SP_Y" + 0.01)) THEN
       #pos_Y_alcanzada := true;
   END_IF;

   IF ("Z" >= ("SP_Z" - 0.01)) AND ("Z" <= ("SP_Z" + 0.01)) THEN
       #pos_Z_alcanzada := true;
   END_IF;
END_FUNCTION

// folder: OBs

ORGANIZATION_BLOCK "Main"   // OB1, LAD, ProgramCycle
TITLE = "Main Program Sweep (Cycle)"
{ S7_Optimized_Access := 'TRUE' }
VERSION : 0.1
   VAR_INPUT
      Initial_Call : Bool;   // Initial call of this OB
      Remanence : Bool;   // =True, if remanent data are available
   END_VAR
   VAR_TEMP   // added for the SCL form of the ladder/FBD networks
      _w1 : Bool;
   END_VAR
BEGIN

REGION Network 1: Funcion necesaria para conexion con factory IO
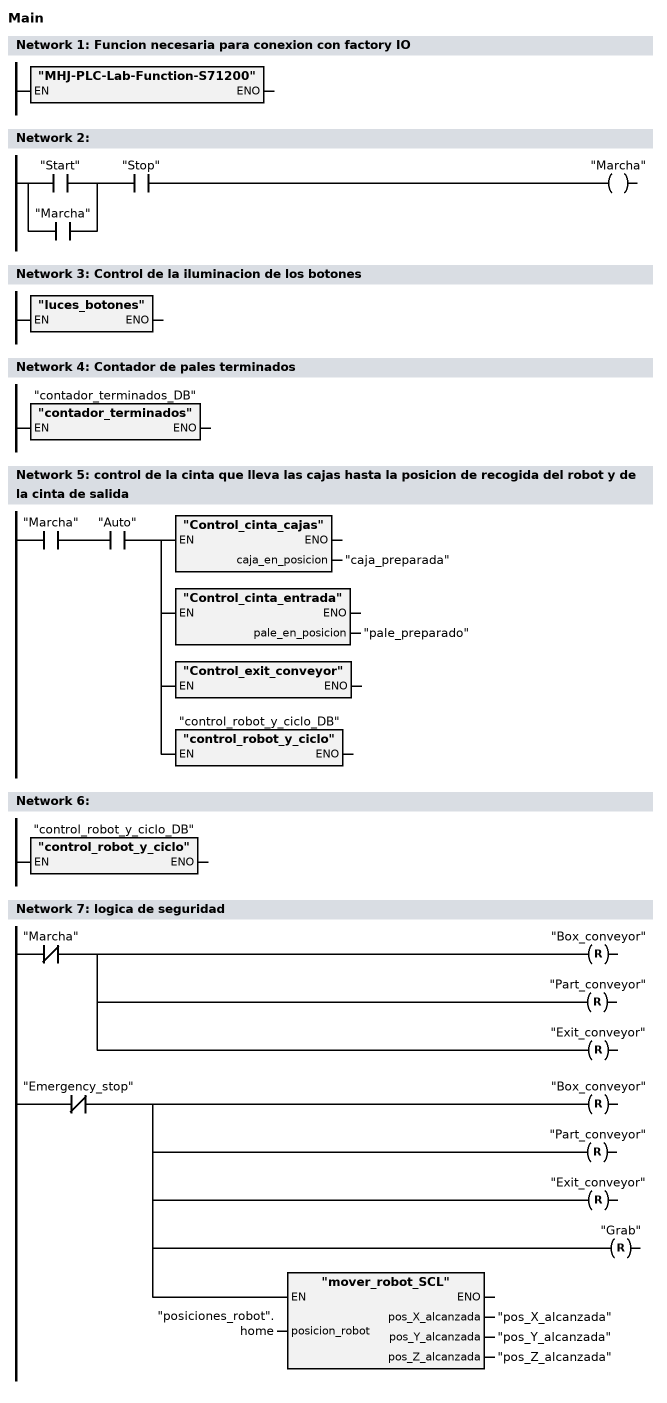
   RUNG wire#powerrail
      "MHJ-PLC-Lab-Function-S71200"()
   END_RUNG
   // the same network as SCL:
   "MHJ-PLC-Lab-Function-S71200"();
END_REGION

REGION Network 2
   RUNG wire#powerrail
      Contact( "Start" )
      wire#w1
      Contact( "Stop" )
      Coil( "Marcha" )
   END_RUNG
   RUNG wire#powerrail
      Contact( "Marcha" )
   END_RUNG wire#w1
   // the same network as SCL:
   "Marcha" := ("Start" OR "Marcha") AND "Stop";
END_REGION

REGION Network 3: Control de la iluminacion de los botones
   RUNG wire#powerrail
      "luces_botones"()
   END_RUNG
   // the same network as SCL:
   "luces_botones"();
END_REGION

REGION Network 4: Contador de pales terminados
   RUNG wire#powerrail
      "contador_terminados_DB"()
   END_RUNG
   // the same network as SCL:
   "contador_terminados_DB"();   // "contador_terminados"
END_REGION

REGION Network 5: control de la cinta que lleva las cajas hasta la posicion de recogida del robot y de la cinta de salida
   RUNG wire#powerrail
      Contact( "Marcha" )
      Contact( "Auto" )
      wire#w1
      "Control_cinta_cajas"(caja_en_posicion => "caja_preparada")
   END_RUNG
   RUNG wire#w1
      "Control_cinta_entrada"(pale_en_posicion => "pale_preparado")
   END_RUNG
   RUNG wire#w1
      "Control_exit_conveyor"()
   END_RUNG
   RUNG wire#w1
      "control_robot_y_ciclo_DB"()
   END_RUNG
   // the same network as SCL:
   #_w1 := "Marcha" AND "Auto";
   IF #_w1 THEN
       "Control_cinta_cajas"(caja_en_posicion => "caja_preparada");
       "Control_cinta_entrada"(pale_en_posicion => "pale_preparado");
       "Control_exit_conveyor"();
       "control_robot_y_ciclo_DB"();   // "control_robot_y_ciclo"
   END_IF;
END_REGION

REGION Network 6
   RUNG wire#powerrail
      "control_robot_y_ciclo_DB"()
   END_RUNG
   // the same network as SCL:
   "control_robot_y_ciclo_DB"();   // "control_robot_y_ciclo"
END_REGION

REGION Network 7: logica de seguridad
   RUNG wire#powerrail
      I_Contact( "Marcha" )
      wire#w1
      R_Coil( "Box_conveyor" )
   END_RUNG
   RUNG wire#w1
      R_Coil( "Part_conveyor" )
   END_RUNG
   RUNG wire#w1
      R_Coil( "Exit_conveyor" )
   END_RUNG
   RUNG wire#powerrail
      I_Contact( "Emergency_stop" )
      wire#w2
      R_Coil( "Box_conveyor" )
   END_RUNG
   RUNG wire#w2
      R_Coil( "Part_conveyor" )
   END_RUNG
   RUNG wire#w2
      R_Coil( "Exit_conveyor" )
   END_RUNG
   RUNG wire#w2
      R_Coil( "Grab" )
   END_RUNG
   RUNG wire#w2
      "mover_robot_SCL"(posicion_robot := "posiciones_robot".home, pos_X_alcanzada => "pos_X_alcanzada", pos_Y_alcanzada => "pos_Y_alcanzada", pos_Z_alcanzada => "pos_Z_alcanzada")
   END_RUNG
   // the same network as SCL:
   IF NOT "Marcha" THEN
       "Box_conveyor" := FALSE;
       "Part_conveyor" := FALSE;
       "Exit_conveyor" := FALSE;
   END_IF;
   IF NOT "Emergency_stop" THEN
       "Box_conveyor" := FALSE;
       "Part_conveyor" := FALSE;
       "Exit_conveyor" := FALSE;
       "Grab" := FALSE;
       "mover_robot_SCL"(posicion_robot := "posiciones_robot".home,
                         pos_X_alcanzada => "pos_X_alcanzada",
                         pos_Y_alcanzada => "pos_Y_alcanzada",
                         pos_Z_alcanzada => "pos_Z_alcanzada");
   END_IF;
END_REGION
END_ORGANIZATION_BLOCK

ORGANIZATION_BLOCK "Valores_de_arranque"   // OB100, LAD, Startup
TITLE = "Complete Restart"
{ S7_Optimized_Access := 'TRUE' }
VERSION : 0.1
   VAR_INPUT
      LostRetentive : Bool;   // True if retentive data are lost
      LostRTC : Bool;   // True if date and time are lost
   END_VAR
BEGIN

REGION Network 1: Cinta para las cajas
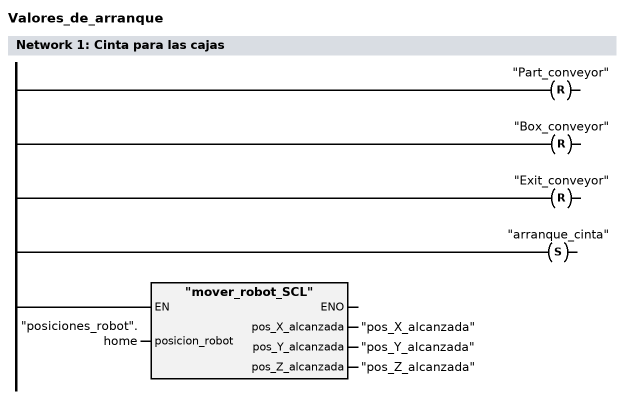
   RUNG wire#powerrail
      R_Coil( "Part_conveyor" )
   END_RUNG
   RUNG wire#powerrail
      R_Coil( "Box_conveyor" )
   END_RUNG
   RUNG wire#powerrail
      R_Coil( "Exit_conveyor" )
   END_RUNG
   RUNG wire#powerrail
      S_Coil( "arranque_cinta" )
   END_RUNG
   RUNG wire#powerrail
      "mover_robot_SCL"(posicion_robot := "posiciones_robot".home, pos_X_alcanzada => "pos_X_alcanzada", pos_Y_alcanzada => "pos_Y_alcanzada", pos_Z_alcanzada => "pos_Z_alcanzada")
   END_RUNG
   // the same network as SCL:
   "Part_conveyor" := FALSE;
   "Box_conveyor" := FALSE;
   "Exit_conveyor" := FALSE;
   "arranque_cinta" := TRUE;
   "mover_robot_SCL"(posicion_robot := "posiciones_robot".home,
                     pos_X_alcanzada => "pos_X_alcanzada",
                     pos_Y_alcanzada => "pos_Y_alcanzada",
                     pos_Z_alcanzada => "pos_Z_alcanzada");
END_REGION
END_ORGANIZATION_BLOCK